(* CODESYS project EAS PLC.library
   Author: EAS
   Placeholder: EAS
   Title: EAS PLC
   Version: 1.0.0
   DefaultNamespace: EAS
   Company: ESCARRE AUTOMATIZACION Y SERVICIOS sl

Project tree, tasks and I/O mapping:
  libraries: Tc2_Standard, * (Beckhoff Automation GmbH); Tc2_System, * (Beckhoff Automation GmbH); Tc3_Module, * (Beckhoff Automation GmbH); Util, * (System)
  DUTs/
    data type TipusCurva
  GVLs/
    global variables GVL
  POUs/
    PLC/
      AddTanks/
        function block Circulation_TK [ST]
        function block Drain_TK [ST]
        function fCurvePerCen [ST]
        function block Introduction [ST]
        function block Introduction_M [ST]
      Elements/
        function block LiterCounter [ST]
        function block LitersPerLevel [ST]
        function block MeterCounter [ST]
        function block PulseTrain [ST]
        function block Washing_HT [ST]
      Fill/
        function block TemperatureFill [ST]
      Utils/
        AnalogConversions/
          function Canvi_Escala [ST]
          function Conv_Temp [ST]
        BitsConversions/
          function block Bits_to_Dword [ST]
          function block Bits_to_word [ST]
          function block Dword_to_bits [ST]
          function block Word_to_bits [ST]
        Counters/
          function block Calcul_Frequencia [ST]
          function block ContadorRapid [ST]
        FreqCycle/
          function block CalcFreq [ST]
          function block TCicle [ST]
        Timers/
          function block TMP [ST]
          function block TMPpausa [ST]
  VISUs/
*)

// DUTs/TipusCurva
TYPE TipusCurva :
STRUCT
	Table:ARRAY [0..10] OF point;
END_STRUCT
END_TYPE

// GVLs/GVL
VAR_GLOBAL RETAIN

(*=======================================	*)
(*		Curvas								*)
(*=======================================	*)

	CurvePerCent:ARRAY[0..19]OF TipusCurva;

END_VAR

// POUs/PLC/AddTanks/Circulation_TK
FUNCTION_BLOCK Circulation_TK
(*****************************************************************
Execute the recirculation of the add tank (Mac -> tank, tank -> mac) - 01/12/2021
v1.00
****************************************************************)
VAR_INPUT
	xActvRecirc:BOOL;				// Activate the function
	xPulsFinRecirc:BOOL;			// Finish the function
	xLowLevelRecirc:BOOL;			// Add tank Low level for the recirculation
	xHighLevelRecirc:BOOL;			// Add tank high level for the recirculation
	xMinimLevel:BOOL;				// Minimum tank level for the recirculation
	dwDrainTime:DWORD;				// Add tank drain time
END_VAR
VAR_OUTPUT
	xFiRecirc:BOOL;					// Recirculate finished
	xFill:BOOL;						// Add tank fill (runback)
	xIntro:BOOL;					// Add tank introduction (transfer)
END_VAR
VAR
	PararRecirculacio: BOOL;
	PararOmplerta: BOOL;
	OmplirEnRecirculacio: BOOL;
	PararIntroducio: BOOL;
	IntroduccioEnRecirculacio: BOOL;
	srPararRecirculacio : SR;
	TempoDescubrirNivBaix: TMP;
	Reircular: BOOL;
	FiBuidatCubeta: BOOL;
	BuidarCubeta: BOOL;
	TEmpoDrenatBuidat: TMP;
	srFiBuidatCubeta : SR;
END_VAR

// *********** Fin recircula por pulsador *****************
srPararRecirculacio(SET1:=xActvRecirc AND  xPulsFinRecirc, RESET:=NOT xActvRecirc , Q1=>PararRecirculacio );

Reircular := xActvRecirc AND NOT PararRecirculacio;

OmplirEnRecirculacio := Reircular AND NOT PararOmplerta;

IntroduccioEnRecirculacio := Reircular AND NOT PararIntroducio;
// ********* Pausa la introduccion si el nivel esta bajo *****************
TempoDescubrirNivBaix(xIN:=Reircular AND xLowLevelRecirc, dwSegons:=5 , xQ=> , dwTsegons=> );
PararIntroducio := NOT TempoDescubrirNivBaix.xQ; 

PararOmplerta := Reircular AND xHighLevelRecirc;

BuidarCubeta := xActvRecirc AND PararRecirculacio;

TEmpoDrenatBuidat(xIN:=BuidarCubeta AND NOT xMinimLevel, dwSegons:=dwDrainTime , xQ=> , dwTsegons=> );

srFiBuidatCubeta(SET1:=TEmpoDrenatBuidat.xQ , RESET:=NOT xActvRecirc , Q1=>FiBuidatCubeta );
// ************ Finaliza la recirculacion ********
xFiRecirc := FiBuidatCubeta;
// ************ Introduz a la maquina **********
xIntro := (BuidarCubeta AND NOT FiBuidatCubeta) OR IntroduccioEnRecirculacio;
// ************ Retorno de bano a la cubeta ********
xFill := OmplirEnRecirculacio;

END_FUNCTION_BLOCK

// POUs/PLC/AddTanks/Introduction
FUNCTION_BLOCK Introduction
(**********************************************************************
Control the transfering and dosing of the add tanks - 01/12/2021
v1.00
***********************************************************************)
VAR_INPUT
	xActvIntro:BOOL;			//Enable the function
	dwCurve:DWORD;				// Dosing curve
	dwTime:DWORD;				// Duration Time
	rLevel:REAL;				// Tank Level
	xLevelMin:BOOL;				// Tank Minimun Level
	xIniCond:BOOL;				// Initial condicions
	xPause:BOOL;				// Pause the function
END_VAR
VAR_OUTPUT
	xFiIntro:BOOL;				// End of the introduction
	rQTeoric:REAL;				// Teoric Quantity of the introduction (%)
	rQreal:REAL;				// Real Quantity of the introduction (%)
	xPrepareIntro:BOOL;			// Prepare an Introduction
	xDosIntro:BOOL;				// Introduct dosing (slow)
	xTransferIntro:BOOL;		// Introduct transfering (fast)
END_VAR
VAR
	IniciarIntro: BOOL;
	TEmpoInici: TMP;
	calculQt: CHARCURVE;
	rampatems: RAMP_REAL;
	tempsreal: REAL;
	Tempsensegons: REAL;
	IntroduccioDosificada: BOOL;
	IntroduccioDirecte: BOOL;
	TempsEnPercentatge: REAL;
	TaulaCurva:ARRAY [0..10]OF point;
	RampaTempsInt: INT;
	QteoricaINT: INT;
	ERROR: BYTE;
	entradaRampa: REAL;

	NivellInicial: REAL;
	TempsNivellinim: TMP;
	FiIntroDosificada: BOOL;
	TempsNivellinimDir: TMP;
	FiDirecte: BOOL;
	srFiIntro :SR;
END_VAR

// Inicia Intro
TEmpoInici(xIN:=xActvIntro AND xIniCond , dwSegons:=2 , xQ=>IniciarIntro , dwTsegons=> );

// Verifica si es introducion directa o dosificada
IF dwTime > 0
	THEN
		IntroduccioDosificada := TRUE;
		IntroduccioDirecte := FALSE;
	ELSE
		IntroduccioDosificada := FALSE;
		IntroduccioDirecte := TRUE;
END_IF

// Calculos del tiempo
Tempsensegons := DWORD_TO_REAL(dwTime*60);

IF IniciarIntro
	THEN
		EntradaRampa := Tempsensegons;
	ELSE
		EntradaRampa := 0;	
		NivellInicial := rLevel;
END_IF

// Si es introducin dosificada calcula la rampa
IF IntroduccioDosificada
	THEN
		rampatems(
			IN:= EntradaRampa, 
			ASCEND:= 1, 
			DESCEND:= Tempsensegons, 
			TIMEBASE:= T#1S, 
			RESET:= (IniciarIntro AND xPause) , 
			OUT=> tempsreal);

		TempsEnPercentatge := (tempsreal/Tempsensegons)*100;
END_IF

RampaTempsInt := REAL_TO_INT(TempsEnPercentatge*100);

TaulaCurva :=  fCurvePerCen(Curve:=DWORD_TO_INT (dwCurve));

calculQt(
	IN:= RampaTempsInt , 
	N:=11 , 
	P:=TaulaCurva , 
	OUT=>QteoricaINT , 
	ERR=>ERROR );

// Si se ha iniciado la introducion calcula el Qreal
IF IniciarIntro AND NivellInicial > 0
	THEN
		rQreal := (rLevel/NivellInicial)*100;
END_IF

rQTeoric := (INT_TO_REAL(QteoricaINT))/100;

xPrepareIntro := IniciarIntro AND NOT xFiIntro;

IF rQreal > rQTeoric AND IniciarIntro AND IntroduccioDosificada AND NOT xFiIntro
	THEN
		xDosIntro := TRUE;
	ELSE
		xDosIntro := FALSE;
END_IF

xTransferIntro := IntroduccioDosificada AND IniciarIntro AND NOT xFiIntro;

TempsNivellinim(xIN:=xLevelMin , dwSegons:=60 , xQ=> , dwTsegons=> );

IF rQTeoric <= 0 OR rQTeoric <= 0 OR TempsNivellinim.xQ OR IntroduccioDosificada OR IniciarIntro OR NOT xLevelMin
	THEN
		FiIntroDosificada := TRUE;
	ELSE
		FiIntroDosificada := FALSE;
END_IF

TempsNivellinimDir(xIN:= NOT xLevelMin , dwSegons:=3 , xQ=> , dwTsegons=> );

FiDirecte := NOT IntroduccioDosificada AND IniciarIntro AND TempsNivellinimDir.xQ;


srFiIntro(SET1:=(FiIntroDosificada OR FiDirecte) AND xActvIntro, RESET:= NOT xActvIntro , Q1=>xFiIntro);

END_FUNCTION_BLOCK

// POUs/PLC/AddTanks/fCurvePerCen
FUNCTION fCurvePerCen : ARRAY [0..10] OF POINT
(*******************************************************
Aquest Bloc Carrega per HardCode els valors de les les Corves percentuals.
Al demanar una corva retorna una taula de punts per a l'introduccio
=========================================
06/09/2006= Error corva7.
********************************************************)
VAR_INPUT
	Curve:INT;			// Curve (0 - 19)
END_VAR

VAR_OUTPUT

END_VAR	

VAR
END_VAR



(*Curve 0*)
GVL.CurvePerCent[0].Table[0].X:=0;
GVL.CurvePerCent[0].Table[0].Y:=10000;
GVL.CurvePerCent[0].Table[1].X:=1000;
GVL.CurvePerCent[0].Table[1].Y:=9000;
GVL.CurvePerCent[0].Table[2].X:=2000;
GVL.CurvePerCent[0].Table[2].Y:=8000;
GVL.CurvePerCent[0].Table[3].X:=3000;
GVL.CurvePerCent[0].Table[3].Y:=7000;
GVL.CurvePerCent[0].Table[4].X:=4000;
GVL.CurvePerCent[0].Table[4].Y:=6000;
GVL.CurvePerCent[0].Table[5].X:=5000;
GVL.CurvePerCent[0].Table[5].Y:=5000;
GVL.CurvePerCent[0].Table[6].X:=6000;
GVL.CurvePerCent[0].Table[6].Y:=4000;
GVL.CurvePerCent[0].Table[7].X:=7000;
GVL.CurvePerCent[0].Table[7].Y:=3000;
GVL.CurvePerCent[0].Table[8].X:=8000;
GVL.CurvePerCent[0].Table[8].Y:=2000;
GVL.CurvePerCent[0].Table[9].X:=9000;
GVL.CurvePerCent[0].Table[9].Y:=1000;
GVL.CurvePerCent[0].Table[10].X:=10000;
GVL.CurvePerCent[0].Table[10].Y:=0;

(*GVL.Curve 1*)
GVL.CurvePerCent[1].Table[0].X:=0;
GVL.CurvePerCent[1].Table[0].Y:=10000;
GVL.CurvePerCent[1].Table[1].X:=1000;
GVL.CurvePerCent[1].Table[1].Y:=9100;
GVL.CurvePerCent[1].Table[2].X:=2000;
GVL.CurvePerCent[1].Table[2].Y:=8200;
GVL.CurvePerCent[1].Table[3].X:=3000;
GVL.CurvePerCent[1].Table[3].Y:=7300;
GVL.CurvePerCent[1].Table[4].X:=4000;
GVL.CurvePerCent[1].Table[4].Y:=6400;
GVL.CurvePerCent[1].Table[5].X:=5000;
GVL.CurvePerCent[1].Table[5].Y:=5400;
GVL.CurvePerCent[1].Table[6].X:=6000;
GVL.CurvePerCent[1].Table[6].Y:=4500;
GVL.CurvePerCent[1].Table[7].X:=7000;
GVL.CurvePerCent[1].Table[7].Y:=3500;
GVL.CurvePerCent[1].Table[8].X:=8000;
GVL.CurvePerCent[1].Table[8].Y:=2400;
GVL.CurvePerCent[1].Table[9].X:=9000;
GVL.CurvePerCent[1].Table[9].Y:=1300;
GVL.CurvePerCent[1].Table[10].X:=10000;
GVL.CurvePerCent[1].Table[10].Y:=0;

(*GVL.Curve 2*)
GVL.CurvePerCent[2].Table[0].X:=0;
GVL.CurvePerCent[2].Table[0].Y:=10000;
GVL.CurvePerCent[2].Table[1].X:=1000;
GVL.CurvePerCent[2].Table[1].Y:=9200;
GVL.CurvePerCent[2].Table[2].X:=2000;
GVL.CurvePerCent[2].Table[2].Y:=8400;
GVL.CurvePerCent[2].Table[3].X:=3000;
GVL.CurvePerCent[2].Table[3].Y:=7600;
GVL.CurvePerCent[2].Table[4].X:=4000;
GVL.CurvePerCent[2].Table[4].Y:=6700;
GVL.CurvePerCent[2].Table[5].X:=5000;
GVL.CurvePerCent[2].Table[5].Y:=5800;
GVL.CurvePerCent[2].Table[6].X:=6000;
GVL.CurvePerCent[2].Table[6].Y:=4900;
GVL.CurvePerCent[2].Table[7].X:=7000;
GVL.CurvePerCent[2].Table[7].Y:=3900;
GVL.CurvePerCent[2].Table[8].X:=8000;
GVL.CurvePerCent[2].Table[8].Y:=2800;
GVL.CurvePerCent[2].Table[9].X:=9000;
GVL.CurvePerCent[2].Table[9].Y:=1500;
GVL.CurvePerCent[2].Table[10].X:=10000;
GVL.CurvePerCent[2].Table[10].Y:=0;

(*GVL.Curve 3*)
GVL.CurvePerCent[3].Table[0].X:=0;
GVL.CurvePerCent[3].Table[0].Y:=10000;
GVL.CurvePerCent[3].Table[1].X:=1000;
GVL.CurvePerCent[3].Table[1].Y:=9300;
GVL.CurvePerCent[3].Table[2].X:=2000;
GVL.CurvePerCent[3].Table[2].Y:=8500;
GVL.CurvePerCent[3].Table[3].X:=3000;
GVL.CurvePerCent[3].Table[3].Y:=7800;
GVL.CurvePerCent[3].Table[4].X:=4000;
GVL.CurvePerCent[3].Table[4].Y:=7000;
GVL.CurvePerCent[3].Table[5].X:=5000;
GVL.CurvePerCent[3].Table[5].Y:=6200;
GVL.CurvePerCent[3].Table[6].X:=6000;
GVL.CurvePerCent[3].Table[6].Y:=5300;
GVL.CurvePerCent[3].Table[7].X:=7000;
GVL.CurvePerCent[3].Table[7].Y:=4400;
GVL.CurvePerCent[3].Table[8].X:=8000;
GVL.CurvePerCent[3].Table[8].Y:=3200;
GVL.CurvePerCent[3].Table[9].X:=9000;
GVL.CurvePerCent[3].Table[9].Y:=1800;
GVL.CurvePerCent[3].Table[10].X:=10000;
GVL.CurvePerCent[3].Table[10].Y:=0;

(*GVL.Curve 4*)
GVL.CurvePerCent[4].Table[0].X:=0;
GVL.CurvePerCent[4].Table[0].Y:=10000;
GVL.CurvePerCent[4].Table[1].X:=1000;
GVL.CurvePerCent[4].Table[1].Y:=9400;
GVL.CurvePerCent[4].Table[2].X:=2000;
GVL.CurvePerCent[4].Table[2].Y:=8600;
GVL.CurvePerCent[4].Table[3].X:=3000;
GVL.CurvePerCent[4].Table[3].Y:=8100;
GVL.CurvePerCent[4].Table[4].X:=4000;
GVL.CurvePerCent[4].Table[4].Y:=7400;
GVL.CurvePerCent[4].Table[5].X:=5000;
GVL.CurvePerCent[4].Table[5].Y:=6600;
GVL.CurvePerCent[4].Table[6].X:=6000;
GVL.CurvePerCent[4].Table[6].Y:=5700;
GVL.CurvePerCent[4].Table[7].X:=7000;
GVL.CurvePerCent[4].Table[7].Y:=4900;
GVL.CurvePerCent[4].Table[8].X:=8000;
GVL.CurvePerCent[4].Table[8].Y:=3600;
GVL.CurvePerCent[4].Table[9].X:=9000;
GVL.CurvePerCent[4].Table[9].Y:=2100;
GVL.CurvePerCent[4].Table[10].X:=10000;
GVL.CurvePerCent[4].Table[10].Y:=0;

(*GVL.Curve 5*)
GVL.CurvePerCent[5].Table[0].X:=0;
GVL.CurvePerCent[5].Table[0].Y:=10000;
GVL.CurvePerCent[5].Table[1].X:=1000;
GVL.CurvePerCent[5].Table[1].Y:=9500;
GVL.CurvePerCent[5].Table[2].X:=2000;
GVL.CurvePerCent[5].Table[2].Y:=8800;
GVL.CurvePerCent[5].Table[3].X:=3000;
GVL.CurvePerCent[5].Table[3].Y:=8300;
GVL.CurvePerCent[5].Table[4].X:=4000;
GVL.CurvePerCent[5].Table[4].Y:=7600;
GVL.CurvePerCent[5].Table[5].X:=5000;
GVL.CurvePerCent[5].Table[5].Y:=7000;
GVL.CurvePerCent[5].Table[6].X:=6000;
GVL.CurvePerCent[5].Table[6].Y:=6200;
GVL.CurvePerCent[5].Table[7].X:=7000;
GVL.CurvePerCent[5].Table[7].Y:=5400;
GVL.CurvePerCent[5].Table[8].X:=8000;
GVL.CurvePerCent[5].Table[8].Y:=4000;
GVL.CurvePerCent[5].Table[9].X:=9000;
GVL.CurvePerCent[5].Table[9].Y:=2300;
GVL.CurvePerCent[5].Table[10].X:=10000;
GVL.CurvePerCent[5].Table[10].Y:=0;

(*GVL.Curve 6*)
GVL.CurvePerCent[6].Table[0].X:=0;
GVL.CurvePerCent[6].Table[0].Y:=10000;
GVL.CurvePerCent[6].Table[1].X:=1000;
GVL.CurvePerCent[6].Table[1].Y:=9500;
GVL.CurvePerCent[6].Table[2].X:=2000;
GVL.CurvePerCent[6].Table[2].Y:=9000;
GVL.CurvePerCent[6].Table[3].X:=3000;
GVL.CurvePerCent[6].Table[3].Y:=8500;
GVL.CurvePerCent[6].Table[4].X:=4000;
GVL.CurvePerCent[6].Table[4].Y:=8000;
GVL.CurvePerCent[6].Table[5].X:=5000;
GVL.CurvePerCent[6].Table[5].Y:=7400;
GVL.CurvePerCent[6].Table[6].X:=6000;
GVL.CurvePerCent[6].Table[6].Y:=6600;
GVL.CurvePerCent[6].Table[7].X:=7000;
GVL.CurvePerCent[6].Table[7].Y:=5800;
GVL.CurvePerCent[6].Table[8].X:=8000;
GVL.CurvePerCent[6].Table[8].Y:=4400;
GVL.CurvePerCent[6].Table[9].X:=9000;
GVL.CurvePerCent[6].Table[9].Y:=2600;
GVL.CurvePerCent[6].Table[10].X:=10000;
GVL.CurvePerCent[6].Table[10].Y:=0;

(*GVL.Curve 7*)
GVL.CurvePerCent[7].Table[0].X:=0;
GVL.CurvePerCent[7].Table[0].Y:=10000;
GVL.CurvePerCent[7].Table[1].X:=1000;
GVL.CurvePerCent[7].Table[1].Y:=9600;
GVL.CurvePerCent[7].Table[2].X:=2000;
GVL.CurvePerCent[7].Table[2].Y:=9200;
GVL.CurvePerCent[7].Table[3].X:=3000;
GVL.CurvePerCent[7].Table[3].Y:=8800;
GVL.CurvePerCent[7].Table[4].X:=4000;
GVL.CurvePerCent[7].Table[4].Y:=8300;
GVL.CurvePerCent[7].Table[5].X:=5000;
GVL.CurvePerCent[7].Table[5].Y:=7800;
GVL.CurvePerCent[7].Table[6].X:=6000;
GVL.CurvePerCent[7].Table[6].Y:=7100;
GVL.CurvePerCent[7].Table[7].X:=7000;
GVL.CurvePerCent[7].Table[7].Y:=6300;
GVL.CurvePerCent[7].Table[8].X:=8000;
GVL.CurvePerCent[7].Table[8].Y:=4800;
GVL.CurvePerCent[7].Table[9].X:=9000;
GVL.CurvePerCent[7].Table[9].Y:=2800;
GVL.CurvePerCent[7].Table[10].X:=10000;
GVL.CurvePerCent[7].Table[10].Y:=0;

(*GVL.Curve 8*)
GVL.CurvePerCent[8].Table[0].X:=0;
GVL.CurvePerCent[8].Table[0].Y:=10000;
GVL.CurvePerCent[8].Table[1].X:=1000;
GVL.CurvePerCent[8].Table[1].Y:=9700;
GVL.CurvePerCent[8].Table[2].X:=2000;
GVL.CurvePerCent[8].Table[2].Y:=9400;
GVL.CurvePerCent[8].Table[3].X:=3000;
GVL.CurvePerCent[8].Table[3].Y:=9100;
GVL.CurvePerCent[8].Table[4].X:=4000;
GVL.CurvePerCent[8].Table[4].Y:=8600;
GVL.CurvePerCent[8].Table[5].X:=5000;
GVL.CurvePerCent[8].Table[5].Y:=8200;
GVL.CurvePerCent[8].Table[6].X:=6000;
GVL.CurvePerCent[8].Table[6].Y:=7500;
GVL.CurvePerCent[8].Table[7].X:=7000;
GVL.CurvePerCent[8].Table[7].Y:=6700;
GVL.CurvePerCent[8].Table[8].X:=8000;
GVL.CurvePerCent[8].Table[8].Y:=5200;
GVL.CurvePerCent[8].Table[9].X:=9000;
GVL.CurvePerCent[8].Table[9].Y:=3100;
GVL.CurvePerCent[8].Table[10].X:=10000;
GVL.CurvePerCent[8].Table[10].Y:=0;

(*GVL.Curve 9*)
GVL.CurvePerCent[9].Table[0].X:=0;
GVL.CurvePerCent[9].Table[0].Y:=10000;
GVL.CurvePerCent[9].Table[1].X:=1000;
GVL.CurvePerCent[9].Table[1].Y:=9800;
GVL.CurvePerCent[9].Table[2].X:=2000;
GVL.CurvePerCent[9].Table[2].Y:=9600;
GVL.CurvePerCent[9].Table[3].X:=3000;
GVL.CurvePerCent[9].Table[3].Y:=9300;
GVL.CurvePerCent[9].Table[4].X:=4000;
GVL.CurvePerCent[9].Table[4].Y:=9000;
GVL.CurvePerCent[9].Table[5].X:=5000;
GVL.CurvePerCent[9].Table[5].Y:=8600;
GVL.CurvePerCent[9].Table[6].X:=6000;
GVL.CurvePerCent[9].Table[6].Y:=7900;
GVL.CurvePerCent[9].Table[7].X:=7000;
GVL.CurvePerCent[9].Table[7].Y:=7100;
GVL.CurvePerCent[9].Table[8].X:=8000;
GVL.CurvePerCent[9].Table[8].Y:=5600;
GVL.CurvePerCent[9].Table[9].X:=9000;
GVL.CurvePerCent[9].Table[9].Y:=3400;
GVL.CurvePerCent[9].Table[10].X:=10000;
GVL.CurvePerCent[9].Table[10].Y:=0;

(*GVL.Curve 10*)
GVL.CurvePerCent[10].Table[0].X:=0;
GVL.CurvePerCent[10].Table[0].Y:=10000;
GVL.CurvePerCent[10].Table[1].X:=1000;
GVL.CurvePerCent[10].Table[1].Y:=9000;
GVL.CurvePerCent[10].Table[2].X:=2000;
GVL.CurvePerCent[10].Table[2].Y:=8000;
GVL.CurvePerCent[10].Table[3].X:=3000;
GVL.CurvePerCent[10].Table[3].Y:=7000;
GVL.CurvePerCent[10].Table[4].X:=4000;
GVL.CurvePerCent[10].Table[4].Y:=6000;
GVL.CurvePerCent[10].Table[5].X:=5000;
GVL.CurvePerCent[10].Table[5].Y:=5000;
GVL.CurvePerCent[10].Table[6].X:=6000;
GVL.CurvePerCent[10].Table[6].Y:=4000;
GVL.CurvePerCent[10].Table[7].X:=7000;
GVL.CurvePerCent[10].Table[7].Y:=3000;
GVL.CurvePerCent[10].Table[8].X:=8000;
GVL.CurvePerCent[10].Table[8].Y:=2000;
GVL.CurvePerCent[10].Table[9].X:=9000;
GVL.CurvePerCent[10].Table[9].Y:=1000;
GVL.CurvePerCent[10].Table[10].X:=10000;
GVL.CurvePerCent[10].Table[10].Y:=0;

(*GVL.Curve 11*)
GVL.CurvePerCent[11].Table[0].X:=0;
GVL.CurvePerCent[11].Table[0].Y:=10000;
GVL.CurvePerCent[11].Table[1].X:=1000;
GVL.CurvePerCent[11].Table[1].Y:=8700;
GVL.CurvePerCent[11].Table[2].X:=2000;
GVL.CurvePerCent[11].Table[2].Y:=7600;
GVL.CurvePerCent[11].Table[3].X:=3000;
GVL.CurvePerCent[11].Table[3].Y:=6500;
GVL.CurvePerCent[11].Table[4].X:=4000;
GVL.CurvePerCent[11].Table[4].Y:=5500;
GVL.CurvePerCent[11].Table[5].X:=5000;
GVL.CurvePerCent[11].Table[5].Y:=4600;
GVL.CurvePerCent[11].Table[6].X:=6000;
GVL.CurvePerCent[11].Table[6].Y:=3600;
GVL.CurvePerCent[11].Table[7].X:=7000;
GVL.CurvePerCent[11].Table[7].Y:=2700;
GVL.CurvePerCent[11].Table[8].X:=8000;
GVL.CurvePerCent[11].Table[8].Y:=1800;
GVL.CurvePerCent[11].Table[9].X:=9000;
GVL.CurvePerCent[11].Table[9].Y:=900;
GVL.CurvePerCent[11].Table[10].X:=10000;
GVL.CurvePerCent[11].Table[10].Y:=0;

(*GVL.Curve 12*)
GVL.CurvePerCent[12].Table[0].X:=0;
GVL.CurvePerCent[12].Table[0].Y:=10000;
GVL.CurvePerCent[12].Table[1].X:=1000;
GVL.CurvePerCent[12].Table[1].Y:=8500;
GVL.CurvePerCent[12].Table[2].X:=2000;
GVL.CurvePerCent[12].Table[2].Y:=7200;
GVL.CurvePerCent[12].Table[3].X:=3000;
GVL.CurvePerCent[12].Table[3].Y:=6100;
GVL.CurvePerCent[12].Table[4].X:=4000;
GVL.CurvePerCent[12].Table[4].Y:=5100;
GVL.CurvePerCent[12].Table[5].X:=5000;
GVL.CurvePerCent[12].Table[5].Y:=4200;
GVL.CurvePerCent[12].Table[6].X:=6000;
GVL.CurvePerCent[12].Table[6].Y:=3300;
GVL.CurvePerCent[12].Table[7].X:=7000;
GVL.CurvePerCent[12].Table[7].Y:=2400;
GVL.CurvePerCent[12].Table[8].X:=8000;
GVL.CurvePerCent[12].Table[8].Y:=1600;
GVL.CurvePerCent[12].Table[9].X:=9000;
GVL.CurvePerCent[12].Table[9].Y:=800;
GVL.CurvePerCent[12].Table[10].X:=10000;
GVL.CurvePerCent[12].Table[10].Y:=0;

(*GVL.Curve 13*)
GVL.CurvePerCent[13].Table[0].X:=0;
GVL.CurvePerCent[13].Table[0].Y:=10000;
GVL.CurvePerCent[13].Table[1].X:=1000;
GVL.CurvePerCent[13].Table[1].Y:=8200;
GVL.CurvePerCent[13].Table[2].X:=2000;
GVL.CurvePerCent[13].Table[2].Y:=6800;
GVL.CurvePerCent[13].Table[3].X:=3000;
GVL.CurvePerCent[13].Table[3].Y:=5600;
GVL.CurvePerCent[13].Table[4].X:=4000;
GVL.CurvePerCent[13].Table[4].Y:=4700;
GVL.CurvePerCent[13].Table[5].X:=5000;
GVL.CurvePerCent[13].Table[5].Y:=3800;
GVL.CurvePerCent[13].Table[6].X:=6000;
GVL.CurvePerCent[13].Table[6].Y:=3000;
GVL.CurvePerCent[13].Table[7].X:=7000;
GVL.CurvePerCent[13].Table[7].Y:=2200;
GVL.CurvePerCent[13].Table[8].X:=8000;
GVL.CurvePerCent[13].Table[8].Y:=1500;
GVL.CurvePerCent[13].Table[9].X:=9000;
GVL.CurvePerCent[13].Table[9].Y:=700;
GVL.CurvePerCent[13].Table[10].X:=10000;
GVL.CurvePerCent[13].Table[10].Y:=0;

(*GVL.Curve 14*)
GVL.CurvePerCent[14].Table[0].X:=0;
GVL.CurvePerCent[14].Table[0].Y:=10000;
GVL.CurvePerCent[14].Table[1].X:=1000;
GVL.CurvePerCent[14].Table[1].Y:=7900;
GVL.CurvePerCent[14].Table[2].X:=2000;
GVL.CurvePerCent[14].Table[2].Y:=6400;
GVL.CurvePerCent[14].Table[3].X:=3000;
GVL.CurvePerCent[14].Table[3].Y:=5100;
GVL.CurvePerCent[14].Table[4].X:=4000;
GVL.CurvePerCent[14].Table[4].Y:=4300;
GVL.CurvePerCent[14].Table[5].X:=5000;
GVL.CurvePerCent[14].Table[5].Y:=3400;
GVL.CurvePerCent[14].Table[6].X:=6000;
GVL.CurvePerCent[14].Table[6].Y:=2600;
GVL.CurvePerCent[14].Table[7].X:=5000;
GVL.CurvePerCent[14].Table[7].Y:=1900;
GVL.CurvePerCent[14].Table[8].X:=8000;
GVL.CurvePerCent[14].Table[8].Y:=1400;
GVL.CurvePerCent[14].Table[9].X:=9000;
GVL.CurvePerCent[14].Table[9].Y:=600;
GVL.CurvePerCent[14].Table[10].X:=10000;
GVL.CurvePerCent[14].Table[10].Y:=0;

(*GVL.Curve 15*)
GVL.CurvePerCent[15].Table[0].X:=0;
GVL.CurvePerCent[15].Table[0].Y:=10000;
GVL.CurvePerCent[15].Table[1].X:=1000;
GVL.CurvePerCent[15].Table[1].Y:=7700;
GVL.CurvePerCent[15].Table[2].X:=2000;
GVL.CurvePerCent[15].Table[2].Y:=6000;
GVL.CurvePerCent[15].Table[3].X:=3000;
GVL.CurvePerCent[15].Table[3].Y:=4600;
GVL.CurvePerCent[15].Table[4].X:=4000;
GVL.CurvePerCent[15].Table[4].Y:=3800;
GVL.CurvePerCent[15].Table[5].X:=5000;
GVL.CurvePerCent[15].Table[5].Y:=3000;
GVL.CurvePerCent[15].Table[6].X:=6000;
GVL.CurvePerCent[15].Table[6].Y:=2400;
GVL.CurvePerCent[15].Table[7].X:=7000;
GVL.CurvePerCent[15].Table[7].Y:=1700;
GVL.CurvePerCent[15].Table[8].X:=8000;
GVL.CurvePerCent[15].Table[8].Y:=1200;
GVL.CurvePerCent[15].Table[9].X:=9000;
GVL.CurvePerCent[15].Table[9].Y:=500;
GVL.CurvePerCent[15].Table[10].X:=10000;
GVL.CurvePerCent[15].Table[10].Y:=0;

(*GVL.Curve 16*)
GVL.CurvePerCent[16].Table[0].X:=0;
GVL.CurvePerCent[16].Table[0].Y:=10000;
GVL.CurvePerCent[16].Table[1].X:=1000;
GVL.CurvePerCent[16].Table[1].Y:=7400;
GVL.CurvePerCent[16].Table[2].X:=2000;
GVL.CurvePerCent[16].Table[2].Y:=5600;
GVL.CurvePerCent[16].Table[3].X:=3000;
GVL.CurvePerCent[16].Table[3].Y:=4200;
GVL.CurvePerCent[16].Table[4].X:=4000;
GVL.CurvePerCent[16].Table[4].Y:=3400;
GVL.CurvePerCent[16].Table[5].X:=5000;
GVL.CurvePerCent[16].Table[5].Y:=2600;
GVL.CurvePerCent[16].Table[6].X:=6000;
GVL.CurvePerCent[16].Table[6].Y:=2000;
GVL.CurvePerCent[16].Table[7].X:=7000;
GVL.CurvePerCent[16].Table[7].Y:=1500;
GVL.CurvePerCent[16].Table[8].X:=8000;
GVL.CurvePerCent[16].Table[8].Y:=1000;
GVL.CurvePerCent[16].Table[9].X:=9000;
GVL.CurvePerCent[16].Table[9].Y:=500;
GVL.CurvePerCent[16].Table[10].X:=10000;
GVL.CurvePerCent[16].Table[10].Y:=0;

(*GVL.Curve 17*)
GVL.CurvePerCent[17].Table[0].X:=0;
GVL.CurvePerCent[17].Table[0].Y:=10000;
GVL.CurvePerCent[17].Table[1].X:=1000;
GVL.CurvePerCent[17].Table[1].Y:=7200;
GVL.CurvePerCent[17].Table[2].X:=2000;
GVL.CurvePerCent[17].Table[2].Y:=5200;
GVL.CurvePerCent[17].Table[3].X:=3000;
GVL.CurvePerCent[17].Table[3].Y:=3700;
GVL.CurvePerCent[17].Table[4].X:=4000;
GVL.CurvePerCent[17].Table[4].Y:=2900;
GVL.CurvePerCent[17].Table[5].X:=5000;
GVL.CurvePerCent[17].Table[5].Y:=2200;
GVL.CurvePerCent[17].Table[6].X:=6000;
GVL.CurvePerCent[17].Table[6].Y:=1700;
GVL.CurvePerCent[17].Table[7].X:=7000;
GVL.CurvePerCent[17].Table[7].Y:=1200;
GVL.CurvePerCent[17].Table[8].X:=8000;
GVL.CurvePerCent[17].Table[8].Y:=800;
GVL.CurvePerCent[17].Table[9].X:=9000;
GVL.CurvePerCent[17].Table[9].Y:=400;
GVL.CurvePerCent[17].Table[10].X:=10000;
GVL.CurvePerCent[17].Table[10].Y:=0;

(*GVL.Curve 18*)
GVL.CurvePerCent[18].Table[0].X:=0;
GVL.CurvePerCent[18].Table[0].Y:=10000;
GVL.CurvePerCent[18].Table[1].X:=1000;
GVL.CurvePerCent[18].Table[1].Y:=6900;
GVL.CurvePerCent[18].Table[2].X:=2000;
GVL.CurvePerCent[18].Table[2].Y:=4800;
GVL.CurvePerCent[18].Table[3].X:=3000;
GVL.CurvePerCent[18].Table[3].Y:=3300;
GVL.CurvePerCent[18].Table[4].X:=4000;
GVL.CurvePerCent[18].Table[4].Y:=2500;
GVL.CurvePerCent[18].Table[5].X:=5000;
GVL.CurvePerCent[18].Table[5].Y:=1800;
GVL.CurvePerCent[18].Table[6].X:=6000;
GVL.CurvePerCent[18].Table[6].Y:=1400;
GVL.CurvePerCent[18].Table[7].X:=7000;
GVL.CurvePerCent[18].Table[7].Y:=900;
GVL.CurvePerCent[18].Table[8].X:=8000;
GVL.CurvePerCent[18].Table[8].Y:=600;
GVL.CurvePerCent[18].Table[9].X:=9000;
GVL.CurvePerCent[18].Table[9].Y:=300;
GVL.CurvePerCent[18].Table[10].X:=10000;
GVL.CurvePerCent[18].Table[10].Y:=0;

(*GVL.Curve 19*)
GVL.CurvePerCent[19].Table[0].X:=0;
GVL.CurvePerCent[19].Table[0].Y:=10000;
GVL.CurvePerCent[19].Table[1].X:=1000;
GVL.CurvePerCent[19].Table[1].Y:=6600;
GVL.CurvePerCent[19].Table[2].X:=2000;
GVL.CurvePerCent[19].Table[2].Y:=4400;
GVL.CurvePerCent[19].Table[3].X:=3000;
GVL.CurvePerCent[19].Table[3].Y:=2900;
GVL.CurvePerCent[19].Table[4].X:=4000;
GVL.CurvePerCent[19].Table[4].Y:=1900;
GVL.CurvePerCent[19].Table[5].X:=5000;
GVL.CurvePerCent[19].Table[5].Y:=1400;
GVL.CurvePerCent[19].Table[6].X:=6000;
GVL.CurvePerCent[19].Table[6].Y:=1000;
GVL.CurvePerCent[19].Table[7].X:=7000;
GVL.CurvePerCent[19].Table[7].Y:=700;
GVL.CurvePerCent[19].Table[8].X:=8000;
GVL.CurvePerCent[19].Table[8].Y:=400;
GVL.CurvePerCent[19].Table[9].X:=9000;
GVL.CurvePerCent[19].Table[9].Y:=200;
GVL.CurvePerCent[19].Table[10].X:=10000;
GVL.CurvePerCent[19].Table[10].Y:=0;


(*************************************************************************************************)
(*	Cargar Curve	*)

fCurvePerCen:=CurvePerCent[Curve].Table;

END_FUNCTION

// POUs/PLC/Utils/Timers/TMP
FUNCTION_BLOCK TMP
(**********************************************************
Timer in seconds with a DWORD input - 29/11/2021
V1.0
*********************************************************)
VAR_INPUT
	xIN:BOOL;			// Enable Input
	dwSegons:DWORD;		// Setpoint Time (seconds) Input
END_VAR
VAR_OUTPUT
	xQ:BOOL;					// Boolean Output
	dwTsegons:DWORD;			// Currently Time (seconds) Output
END_VAR

VAR
	TEmporitz: TON;
	Temps: TIME;
	TempsTrans: TIME;
END_VAR

Temps := REAL_TO_TIME (DWORD_TO_REAL (dwSegons)*1000);

TEmporitz(IN:=xIN , PT:=Temps , Q=>xQ , ET=>TempsTrans );

dwTsegons := REAL_TO_DWORD(TIME_TO_REAL (TempsTrans)/1000);

END_FUNCTION_BLOCK

// POUs/PLC/AddTanks/Drain_TK
FUNCTION_BLOCK Drain_TK 
(*************************************************************++
Execute the washing and drain of an add tank.
Available drain options:
type=0 => all the washings (2 to machine + 1 to the drain), 
type=1 => 1 to the machine,
type=2 => 2 to the machine,
type=3 => (2 to machine + 1 to the drain), 
01/12/2021
V1.00
*******************************************************************)
VAR_INPUT
	xStartWash:BOOL;			// Enable function input
	xMinimLevel:BOOL;			// Minimum Level Input
	dwDetectLowLevelTime:DWORD;	// Delay to detect the low level
	dwDrainTime:DWORD;			// Drain Time
	dw1stWashTime:DWORD;		// 1st Wash Time
	dw2ndWashTime:DWORD;		// 2nd Wash Time
	dw3rdWashTime:DWORD;		// 3rd Wash Time
	DrainType:DWORD;			// Drain Option (0 - 3)
END_VAR

VAR_OUTPUT
	xFinWash:BOOL;				// Function finished			
	xWash:BOOL;					// Fill the add tank output
	xToMachine:BOOL;			// Transfer add tank to machine
	xToDrain:BOOL;				// Drain add tank
END_VAR

VAR
	FerTotsElsRentats: BOOL;
	NomesRentatsAMaquina: BOOL;
	NoFerRentats: BOOL;
	FiPrimerRentat: BOOL;
	PrimerRentat: BOOL;
	TempoPrimerRentat: TMP;
	FiPrimerBuidat: BOOL;
	PrimerBuidat: BOOL;
	FiSegonRentat: BOOL;
	SegonRentat: BOOL;
	FiSegonBuidat: BOOL;
	SegonBuidat: BOOL;
	TempoPrimerBuidat: TMP;
	TempoSegonRentat: TMP;
	TempoSegonBuidat: TMP;
	TempoTercerRentat: TMP;
	TempoTercerBuidat: TMP;
	FiTercerRentat: BOOL;
	TercerRentat: BOOL;
	FiTercerBuidat: BOOL;
	TercerBuidat: BOOL;
	TempoBuit: TMP;
	ComencaArentar: BOOL;
	BuidaDelTot: BOOL;
	srComencaArentar : SR;
	srFiPrimerRentat : SR;
	srFiPrimerBuidat : SR;
	srFiSegonRentat  : SR;
	srFiSegonBuidat  : SR;
	srFiTercerRentat : SR;
	srFiTercerBuidat : SR;
END_VAR

// ********** Define el tipo de lavado ***********
CASE DrainType OF
	0 : FerTotsElsRentats := TRUE;
		NoFerRentats := FALSE;
		NomesRentatsAMaquina := FALSE;
	1 : FerTotsElsRentats := FALSE;
		NoFerRentats := TRUE;
		NomesRentatsAMaquina := FALSE;
	2 : FerTotsElsRentats := FALSE;
		NoFerRentats := FALSE;
		NomesRentatsAMaquina := TRUE;
	3 : FerTotsElsRentats := TRUE;
		NoFerRentats := FALSE;
		NomesRentatsAMaquina := FALSE;
END_CASE

// ************** Empeza el lavado **************
TempoBuit(xIN:=xStartWash AND NOT  xMinimLevel, dwSegons:=2 , xQ=> , dwTsegons=> );
srComencaArentar(SET1:=TempoBuit.xQ , RESET:= NOT xStartWash , Q1=>ComencaArentar );

BuidaDelTot := xStartWash AND NOT ComencaArentar;

// ********** Control Primer Lavado ******************
PrimerRentat := ComencaArentar AND NOT FiPrimerRentat;

TempoPrimerRentat(xIN:=ComencaArentar , dwSegons:=dw1stWashTime , xQ=> , dwTsegons=> );
srFiPrimerRentat(SET1:=TempoPrimerRentat.xQ , RESET:= NOT xStartWash , Q1=>FiPrimerRentat );

PrimerBuidat := FiPrimerRentat AND NOT FiPrimerBuidat;

TempoPrimerBuidat(xIN:=PrimerBuidat AND NOT  xMinimLevel, dwSegons:=dwDetectLowLevelTime , xQ=> , dwTsegons=> );
srFiPrimerBuidat(SET1:=TempoPrimerBuidat.xQ , RESET:=NOT xStartWash  , Q1=>FiPrimerBuidat );

// ********** Control Segun Lavado ***************** 
SegonRentat := FiPrimerBuidat AND NOT FiSegonRentat;

TempoSegonRentat(xIN:=SegonRentat , dwSegons:=dw2ndWashTime , xQ=> , dwTsegons=> );
srFiSegonRentat(SET1:=TempoSegonRentat.xQ , RESET:=NOT xStartWash  , Q1=>FiSegonRentat );

SegonBuidat := FiSegonRentat AND NOT FiSegonBuidat;

TempoSegonBuidat(xIN:=SegonBuidat AND NOT xMinimLevel, dwSegons:=dwDetectLowLevelTime , xQ=> , dwTsegons=> );
srFiSegonBuidat(SET1:=TempoSegonBuidat.xQ , RESET:=NOT xStartWash  , Q1=>FiSegonBuidat );

// ********** Control Tercer Lavado ***************** 
TercerRentat := FiSegonBuidat AND NOT FiTercerRentat;

TempoTercerRentat(xIN:=TercerRentat , dwSegons:=dw3rdWashTime , xQ=> , dwTsegons=> );
srFiTercerRentat(SET1:=TempoTercerRentat.xQ , RESET:=NOT xStartWash  , Q1=>FiTercerRentat );

TercerBuidat := FiTercerRentat AND NOT FiTercerBuidat;

TempoTercerBuidat(xIN:=TercerBuidat AND NOT xMinimLevel, dwSegons:=dwDrainTime , xQ=> , dwTsegons=> );
srFiTercerBuidat(SET1:=TempoTercerBuidat.xQ , RESET:=NOT xStartWash  , Q1=>FiTercerBuidat);

// ************* Finaliza los lavados ****************
xFinWash := xStartWash AND ((FerTotsElsRentats AND FiTercerBuidat) OR (NomesRentatsAMaquina AND FiSegonBuidat) OR (NoFerRentats AND FiPrimerBuidat));

// ************** Activa salidas *************
xWash	:= xStartWash AND (PrimerRentat OR SegonRentat OR TercerRentat);

xToMachine := NOT xFinWash AND (PrimerBuidat OR SegonBuidat OR BuidaDelTot);

xToDrain := NOT xFinWash AND TercerBuidat;

END_FUNCTION_BLOCK

// POUs/PLC/AddTanks/Introduction_M
FUNCTION_BLOCK Introduction_M
(**********************************************************************
Control the transfering and dosing of the add tanks with proportional valve
- 01/12/2021
v1.00
***********************************************************************)
VAR_INPUT
	xActvIntro:BOOL;			//Enable the function
	dwCurve:DWORD;				// Dosing curve
	dwTime:DWORD;				// Duration Time
	rLevel:REAL;				// Tank Level
	xLevelMin:BOOL;				// Tank Minimun Level
	xIniCond:BOOL;				// Initial condicions
	xPause:BOOL;				// Pause the function
	rPro: REAL;					// PID - P
	rInt: REAL;					// PID - I
	rDer: REAL;					// PID - D
END_VAR
VAR_OUTPUT
	xFiIntro:BOOL;				// End of the introduction
	rQTeoric:REAL;				// Teoric Quantity of the introduction (%)
	rQreal:REAL;				// Real Quantity of the introduction (%)
	xPrepareIntro:BOOL;			// Prepare an Introduction
	xDosIntro:BOOL;				// Introduct dosing (slow)
	xTransferIntro:BOOL;		// Introduct transfering (fast)
	rProportionalValve:REAL;	// % open proportiuonal valve
END_VAR
VAR
	IniciarIntro: BOOL;
	TEmpoInici: TMP;

	calculQt: CHARCURVE;
	rampatems: RAMP_REAL;
	tempsreal: REAL;
	Tempsensegons: REAL;

	IntroduccioDosificada: BOOL;
	IntroduccioDirecte: BOOL;
	TempsEnPercentatge: REAL;
	TaulaCurva:ARRAY [0..10]OF point;
	RampaTempsInt: INT;
	QteoricaINT: INT;
	ERROR: BYTE;
	entradaRampa: REAL;
	NivellInicial: REAL;
	TempsNivellinim: TMP;
	FiIntroDosificada: BOOL;
	TempsNivellinimDir: TMP;
	FiDirecte: BOOL;
	AperturaValvRegulant: PID;
	srFiIntro :SR;
	APERTURApid: REAL;
END_VAR

// *********** Inicia Intro ********************
TEmpoInici(xIN:=xActvIntro AND xIniCond , dwSegons:=2 , xQ=>IniciarIntro , dwTsegons=> );

// ************ Verifica si es introducion directa o dosificada *****************
IF dwTime > 0
	THEN
		IntroduccioDosificada := TRUE;
		IntroduccioDirecte := FALSE;
	ELSE
		IntroduccioDosificada := FALSE;
		IntroduccioDirecte := TRUE;
END_IF

// *************** Calculos del tiempo **********************
Tempsensegons := DWORD_TO_REAL(dwTime*60);

IF IniciarIntro
	THEN
		EntradaRampa := Tempsensegons;
	ELSE
		EntradaRampa := 0;	
		NivellInicial := rLevel;
END_IF

// ************* Si es introducin dosificada calcula la rampa *************
IF IntroduccioDosificada
	THEN
		rampatems(
			IN:= EntradaRampa, 
			ASCEND:= 1, 
			DESCEND:= Tempsensegons, 
			TIMEBASE:= T#1S, 
			RESET:= (IniciarIntro AND xPause) , 
			OUT=> tempsreal);

		TempsEnPercentatge := (tempsreal/Tempsensegons)*100;
END_IF

RampaTempsInt := REAL_TO_INT(TempsEnPercentatge*100);

TaulaCurva :=  fCurvePerCen(Curve:=DWORD_TO_INT (dwCurve));

calculQt(
	IN:= RampaTempsInt , 
	N:=11 , 
	P:=TaulaCurva , 
	OUT=>QteoricaINT , 
	ERR=>ERROR );

// **************** Si se ha iniciado la introducion calcula el Qreal *************
IF IniciarIntro AND NivellInicial > 0
	THEN
		rQreal := (rLevel/NivellInicial)*100;
END_IF

rQTeoric := (INT_TO_REAL(QteoricaINT))/100;

xPrepareIntro := IniciarIntro AND NOT xFiIntro;

xDosIntro := IntroduccioDosificada AND IniciarIntro AND NOT xFiIntro;

xTransferIntro := IntroduccioDirecte AND IniciarIntro AND NOT xFiIntro;

TempsNivellinim(xIN:=xLevelMin , dwSegons:=60 , xQ=> , dwTsegons=> );

IF (rQTeoric <= 0 OR rQTeoric <= 0 OR TempsNivellinim.xQ) AND IntroduccioDosificada AND IniciarIntro
	THEN
		FiIntroDosificada := TRUE;
	ELSE
		FiIntroDosificada := FALSE;
END_IF

TempsNivellinimDir(xIN:= NOT xLevelMin , dwSegons:=3 , xQ=> , dwTsegons=> );

FiDirecte := NOT IntroduccioDosificada AND IniciarIntro AND TempsNivellinimDir.xQ;

srFiIntro(SET1:=(FiIntroDosificada OR FiDirecte) AND xActvIntro, RESET:= NOT xActvIntro , Q1=>xFiIntro);

// ************** Regula la apertura de la valvula modulante ****************
AperturaValvRegulant(
	ACTUAL:= 100-rQreal, 
	SET_POINT:= 100-rQTeoric, 
	KP:= rPro, 
	TN:= rInt, 
	TV:= rDer, 
	Y_MANUAL:= , 
	Y_OFFSET:= , 
	Y_MIN:= 0, 
	Y_MAX:= 100, 
	MANUAL:= , 
	RESET:= NOT xDosIntro OR AperturaValvRegulant.OVERFLOW , 
	Y=> rProportionalValve, 
	LIMITS_ACTIVE=> , 
	OVERFLOW=> );

END_FUNCTION_BLOCK

// POUs/PLC/Elements/LiterCounter
FUNCTION_BLOCK LiterCounter
(*************************************************************
Convert a flow input into liters - 01/12/2021
V1.00
*************************************************************)
VAR_INPUT
	xActive : BOOL;			// Active the function
	rFlow :   REAL;			// Flow Input (l/min)
END_VAR
VAR_OUTPUT
	rLiters :   REAL;		// Liter output (REAL)
	dwLiters : 	DWORD;		//	Liter output (DDWORD)
END_VAR
VAR
	LitersSum : REAL;
	Periodecicle:Tcicle;
	ov: BOOL;
	INTEG: INTEGRAL;	
END_VAR


INTEG(
	IN:=rFlow , 
	TM:=10 , 
	RESET:=ov OR NOT xActive , 
	OUT=> LitersSum, 
	OVERFLOW=>ov );
	
rLiters := LitersSum/60;
dwLiters := REAL_TO_DWORD(LitersSum/60);

END_FUNCTION_BLOCK

// POUs/PLC/Utils/FreqCycle/TCicle
FUNCTION_BLOCK Tcicle
(**********************************************************
 - 29/11/2021
V1.00
*********************************************************)
VAR_INPUT

END_VAR
VAR_OUTPUT
	dwPeriode_Cicle:DWORD;		// Cycle Peryod
END_VAR

VAR_IN_OUT

END_VAR

VAR
	tempo: TON;
	reset: BOOL;
	t_actual: TIME;
	t_anterior: TIME;
	Periode: TIME;
END_VAR

tempo(IN:=NOT reset , PT:=T#7D , Q=>reset , ET=>t_actual );

Periode:= T_actual-T_anterior;

IF	NOT reset
	THEN
		T_anterior := T_actual;
END_IF

dwPeriode_cicle := TIME_TO_DWORD(Periode);

END_FUNCTION_BLOCK

// POUs/PLC/Elements/LitersPerLevel
FUNCTION_BLOCK LitersPerLevel
(**********************************************
Convert an Level input into Liters - 01/12/2021
V1.00
***********************************************)
VAR_INPUT
	rLevel:REAL;
	dwN0:DWORD;
	dwN10:DWORD;
	dwN20:DWORD;
	dwN30:DWORD;
	dwN40:DWORD;
	dwN50:DWORD;
	dwN60:DWORD;
	dwN70:DWORD;
	dwN80:DWORD;
	dwN90:DWORD;
	dwN100:DWORD;
END_VAR
VAR_OUTPUT
	rLiters:REAL;
END_VAR
VAR
	iLiters:INT;
	LitrosMaq: CHARCURVE;
	litrosNivell:ARRAY[0..10]OF point;
END_VAR


litrosNivell[0].X := 0;
litrosNivell[0].Y := dwN0;
litrosNivell[1].X := 100;
litrosNivell[1].Y := dwN10;
litrosNivell[2].X := 200;
litrosNivell[2].Y := dwN20;
litrosNivell[3].X := 300; 
litrosNivell[3].Y := dwN30;
litrosNivell[4].X := 400;
litrosNivell[4].Y := dwN40;
litrosNivell[5].X := 500;
litrosNivell[5].Y := dwN50;
litrosNivell[6].X := 600;
litrosNivell[6].Y := dwN60;
litrosNivell[7].X := 700;
litrosNivell[7].Y := dwN70;
litrosNivell[8].X := 800;
litrosNivell[8].Y := dwN80;
litrosNivell[9].X := 900;
litrosNivell[9].Y := dwN90;
litrosNivell[10].X := 1000;
litrosNivell[10].Y := dwN100;

LitrosMaq(
	IN:= REAL_TO_INT(rLevel*10) , 
	N:= 11, 
	P:= litrosNivell, 
	OUT=> iLiters, 
	ERR=> );

rLiters := INT_TO_REAL (iLiters);

END_FUNCTION_BLOCK

// POUs/PLC/Elements/MeterCounter
FUNCTION_BLOCK MeterCounter
(*************************************************************
Convert an speed input into meters - 01/12/2021
V1.00
*************************************************************)
VAR_INPUT
	xMachineRunning:BOOL;
	xFabricPresence:BOOL;
	xReset:BOOL;
	rSpeed:REAL;
END_VAR
VAR_OUTPUT
	rMeters:REAL;
END_VAR
VAR
	ContarMetros: BOOL;
	Acumulador: ContadorRapid;
	cumulado: BOOL;
	acumulado: REAL;
	acumuladoInicial: REAL;
	acumuladofinal: REAL;
	Pulsocontador: F_TRIG;
	Acumular: BOOL;
END_VAR

ContarMetros := xMachineRunning AND xFabricPresence;

Pulsocontador(CLK:=ContarMetros , Q=>Acumular);

IF Acumular
	THEN
		acumuladoInicial := acumuladofinal;
END_IF

IF xReset
	THEN
		acumuladoInicial :=0;
		acumuladofinal :=0;
END_IF

Acumulador(bActivate:=ContarMetros AND NOT xReset , rFequency:=rSpeed , rCounter_REAL=>acumulado , dwCounter_DWORD=> );

acumuladofinal := acumulado + acumuladoInicial;

rMeters := acumuladofinal/60;

END_FUNCTION_BLOCK

// POUs/PLC/Utils/Counters/ContadorRapid
FUNCTION_BLOCK ContadorRapid
(**********************************************************
Creat an totalizer from an frequency input - 26/11/2021
V1.00
*********************************************************)
VAR_INPUT
	bActivate:BOOL;			// Start executing the function
	rFequency:REAL;			// Input Frequency
END_VAR

VAR_OUTPUT
	rCounter_REAL:REAL;
	dwCounter_DWORD:DWORD;
END_VAR

VAR
	Periodecicle:Tcicle;
	ov: BOOL;
	INTEG: INTEGRAL;
END_VAR



INTEG(
	IN:=rFequency , 
	TM:=Periodecicle.dwPeriode_Cicle , 
	RESET:= ov OR NOT bActivate , 
	OUT=> rCounter_REAL, 
	OVERFLOW=> ov);

dwCounter_DWORD := REAL_TO_DWORD(rCounter_REAL);

END_FUNCTION_BLOCK

// POUs/PLC/Elements/PulseTrain
FUNCTION_BLOCK PulseTrain
(******************************************************
Generate a Pulse Train based on a % input - 10/12/2021
V1.00
*******************************************************)
VAR_INPUT
	rPorcentatge:REAL;			// Percentual Input (0-100%)
	rPeriode_seg:REAL;			// Period Input (sec)
	rPols_min_ms:REAL;			// Minimum duration of the pulse output (ms)
END_VAR

VAR_OUTPUT
	xT_Pulsos:BOOL;				// Pulse Output
END_VAR

VAR
	PararTren: BOOL;
	SegonsOFFtime: TIME;
	SegonsONtime: TIME;
	SegonsONreal: REAL;
	SegonsOFFreal: REAL;
	AperturaPulso: REAL;
	SegonsCicles: REAL;
	Tiemposinsenal: TMP;
	tempsmin: TIME;
	toff: TON;
	TON: TON;
	PulsMin : BOOL;
	TPulsMin:TP;
END_VAR

AperturaPulso := rPorcentatge;
SegonsCicles := rPeriode_seg;

SegonsONreal := (SegonsCicles*AperturaPulso)/100;
SegonsOFFreal := SegonsCicles-SegonsONreal;

SegonsONtime := REAL_TO_TIME(SegonsONreal*1000);
SegonsOFFtime := REAL_TO_TIME(SegonsOFFreal*1000);

IF SegonsONreal = 0
	THEN
		Tiemposinsenal.xIN := TRUE;
	ELSE
		Tiemposinsenal.xIN := FALSE;
END_IF

Tiemposinsenal(xIN:= , dwSegons:=5 , xQ=>PararTren , dwTsegons=> );
tempsmin := REAL_TO_TIME (rPols_min_ms);

// Generador de pulsos
toff(IN:= NOT ton.Q, PT:=SegonsOFFtime , Q=> , ET=> );
ton(IN:= toff.Q, PT:=SegonsONtime , Q=> , ET=> );

// Utiliza el pulso minimo si el tON es mas pequeno que el pulso minimo
IF SegonsONreal <= rPols_min_ms/1000
	THEN
		PulsMin := TRUE;
	ELSE
		PulsMin := FALSE;
END_IF

TPulsMin(IN:=PulsMin AND  toff.Q, PT:=tempsmin , Q=> , ET=> );

xT_Pulsos := (toff.Q AND NOT PararTren) OR (PulsMin AND TPulsMin.Q);

END_FUNCTION_BLOCK

// POUs/PLC/Elements/Washing_HT
FUNCTION_BLOCK Washing_HT
(**************************************************************
Execute a continuos washing in high temperature - 01/12/2021
V1.00
***************************************************************)
VAR_INPUT
	xStartDrain : BOOL;					// Enable the function
	xDirectDrain:BOOL;					// Enable direct drain input
	dwTimeFillAuxTank: DWORD;			// Time to transfer from machine to auxiliar tank
	dwTimeCloseAuxTank:DWORD;			// Time to finish the transfering to the auxiliar tank
	dwTimeDepAuxTank:DWORD;				// Time do depressurize auxiliar tank
	dwTimeDrainAunxTank:DWORD;			// Time to drain the auxiliar tank
	dwTimeCloseDrainAuxTank:DWORD;		// Time to garantee that the drain valve has closed
	xAlarmPauseWash:BOOL;				// Alarm Input to stop the function
	
END_VAR

VAR_OUTPUT
	xFillAuxTank:BOOL;					// Transfer from machuine to auxiliar tank
	xDepAuxTank:BOOL;					// depressurize auxiliar tank
	xDrainAuxTank:BOOL;					// Drain auxiliar tank
END_VAR

VAR
	ObrirBuidatRBB: BOOL;
	TempoPas1: TMP;
	TempoPas2: TMP;
	ObrirDespresuritzaRBB: BOOL;
	TempoPas3: TMP;
	ObrirOmplertaRBB: BOOL;
	TancarOmpertaRBB: BOOL;
	TancarBuidatRBB: BOOL;
	FiSequenciaRBB: BOOL;
	TempoPas4: TMP;
	TempoPas5: TMP;
	TemoDespesuritzaRBB: TMP;
	RBBsensePresio: BOOL;
	ObrirRespiraderoRBB: BOOL;
	FiBuidatRBB: BOOL;
	FiBuidatDirecte: F_TRIG;
	PolsFiBuidat: BOOL;
	TempSfINAL: TMP;
	ObrirBuidatAlBuidat: BOOL;
	srObrirOmplertaRBB :SR;
	srObrirRespiraderoRBB:SR;
	srPolsFiBuidat:SR;
	rtBuidatDirecte:F_TRIG;
	
	
END_VAR

// **************** Inicia el ciclo **************************
srObrirOmplertaRBB(SET1:= xStartDrain AND NOT srObrirOmplertaRBB.Q1 , RESET:=xAlarmPauseWash OR (FiSequenciaRBB AND ObrirOmplertaRBB) , Q1=>ObrirOmplertaRBB );


// **************** Temps por cada pas ************************
TempoPas1(xIN:=ObrirOmplertaRBB , dwSegons:=dwTimeFillAuxTank , xQ=>TancarOmpertaRBB , dwTsegons=> );

TempoPas2(xIN:=TancarOmpertaRBB , dwSegons:=dwTimeCloseAuxTank , xQ=>ObrirDespresuritzaRBB , dwTsegons=> );

TempoPas3(xIN:=ObrirDespresuritzaRBB , dwSegons:=dwTimeDepAuxTank , xQ=>ObrirBuidatRBB , dwTsegons=> );

TempoPas4(xIN:=ObrirBuidatRBB , dwSegons:=dwTimeDrainAunxTank , xQ=>TancarBuidatRBB , dwTsegons=> );

TempoPas5(xIN:=TancarBuidatRBB , dwSegons:=dwTimeCloseDrainAuxTank , xQ=>FiSequenciaRBB , dwTsegons=> );


srObrirRespiraderoRBB(SET1:=xDirectDrain AND NOT srObrirRespiraderoRBB.Q1, RESET:=xAlarmPauseWash OR (FiBuidatRBB AND ObrirRespiraderoRBB) , Q1=>ObrirRespiraderoRBB );

TemoDespesuritzaRBB(xIN:=ObrirRespiraderoRBB , dwSegons:=dwTimeDepAuxTank , xQ=>RBBsensePresio , dwTsegons=> );

rtBuidatDirecte(CLK:=xDirectDrain , Q=> );
srPolsFiBuidat(SET1:=rtBuidatDirecte.Q , RESET:=FiBuidatRBB , Q1=>PolsFiBuidat );

TempSfINAL(xIN:=PolsFiBuidat , dwSegons:=5 , xQ=>FiBuidatRBB , dwTsegons=> );

ObrirBuidatAlBuidat := xDirectDrain AND NOT FiBuidatRBB;

///*************************** Activa salidas ******************************
xFillAuxTank := (ObrirOmplertaRBB AND NOT TancarOmpertaRBB AND NOT xAlarmPauseWash) OR (xDirectDrain AND RBBsensePresio);

xDepAuxTank := (ObrirDespresuritzaRBB AND NOT TancarBuidatRBB AND NOT xAlarmPauseWash) OR xDirectDrain;

xDrainAuxTank := (ObrirBuidatRBB AND NOT TancarBuidatRBB AND NOT xAlarmPauseWash) OR ObrirBuidatAlBuidat;

END_FUNCTION_BLOCK

// POUs/PLC/Fill/TemperatureFill
FUNCTION_BLOCK TemperatureFill
(**********************************************************
Fill with a Temperature SetPoint - 30/11/2021
V1.00
*********************************************************)
VAR_INPUT
	xActiv			:	BOOL;		//Enable the temperature control
	rTempSP			:	REAL;		// Temperature SetPoint
	rTempPV			:	REAL;		// Real Temperature 
	rDBHigh			:	REAL;		// Superior DeadBand 
	rDBLow			:	REAL;		// Inferior DeadBand 
	timMaxTime		:	TIME;		//	Maximum time for adjust the temperature
	dwConfigMaxTime:	DWORD;		//	Maximum time configure (1 - Open just cold water, 0 - Open cold and hot water, 2 - Activate Alarm)
	xLevel			:	BOOL;		// Minimum level input
	dwConfigLevel	:	DWORD;		// Level Configure (0 - Disable, 1 - Starts filing with CW and HW, 2 - Starts filing with CW, 3 - Starts filing with HW) 
	timControl		:	TIME;		// Time delay for start adjusting the teperature.
END_VAR
VAR_OUTPUT
	xCWater				:	BOOL;	// Cold Water Output
	xHWater				:	BOOL;	// Hot Water Output
	xAlarmMaxTime		:	BOOL;	// Maximum time alarm Output
END_VAR
VAR
	TempIni 			:	TON;	
	MaxTemp 			:	TON;
	TemperMin			:	REAL;		// Temperatura mínima SP-DBmin	
	TemperMax			:	REAL;		// Temperatura mínima SP+DBmax
		
	CtrlNivel: BOOL;
END_VAR

MaxTemp(IN:=xActiv AND (rTempPV < TemperMin OR rTempPV > TemperMax) AND TempIni.Q AND SEL(CtrlNivel, 1,xLevel)  , PT:=timMaxTime , Q=>xAlarmMaxTime , ET=> );
TempIni(IN:=xActiv, PT:=timControl , Q=> , ET=> );

TemperMax := rTempSP + rDBHigh;
TemperMin := rTempSP - rDBLow;

IF dwConfigLevel > 0
	THEN
		CtrlNivel := TRUE;
	ELSE
		CtrlNivel := FALSE;
END_IF
	

IF xActiv
	THEN
		IF (rTempPV < TemperMax AND rTempPV > TemperMin AND NOT MaxTemp.Q) OR (MaxTemp.Q AND dwConfigMaxTime = 0 AND dwConfigMaxTime <> 2) OR NOT TempIni.Q OR (dwConfigLevel = 1 AND NOT xLevel) 
			THEN
				xCWater :=TRUE;
				xHWater :=TRUE;
		END_IF	
		IF rTempPV > TemperMax AND NOT MaxTemp.Q AND TempIni.Q OR (MaxTemp.Q AND dwConfigMaxTime = 1 AND dwConfigMaxTime <> 2) OR (dwConfigLevel = 3 AND NOT xLevel)
			THEN			
				xCWater :=TRUE;
				xHWater :=FALSE;			
		END_IF 
		IF rTempPV < TemperMin AND NOT MaxTemp.Q AND TempIni.Q OR (dwConfigLevel = 2 AND NOT xLevel)
			THEN			
				xCWater :=FALSE;
				xHWater :=TRUE;			
		END_IF
		IF MaxTemp.Q AND dwConfigMaxTime = 2
			THEN
				xCWater :=FALSE;
				xHWater :=FALSE;
		END_IF
	 ELSE
		xCWater :=FALSE;
		xHWater :=FALSE;			
END_IF

END_FUNCTION_BLOCK

// POUs/PLC/Utils/AnalogConversions/Canvi_Escala
FUNCTION Canvi_Escala:REAL
(**************************************************************
Execute an SCALE from an input value (REAL). If not defined
 the scales, the default values are going to be 0 (min) and 100 (max)
for both, input and output. 26/11/2021
V1.00
***************************************************************)
VAR_INPUT
	rIn:REAL;						// Input Variable
	rIn_Min:REAL:=0;				// Input Low Value
	rIn_Max:REAL:=100;				// Input High Value
	rOut_Min:REAL:=0;				// Output Low Value
	rOut_Max:REAL:=100;				// Output High Value
END_VAR

VAR
	Din: REAL;
	Dout: REAL;
END_VAR

IF rin<rin_Min
	THEN
		rin:=rin_min;
END_IF
IF rin>rin_Max
	THEN
		rin:=rin_max;
END_IF

Din:=rIn_Max-rIn_Min;

IF Din=0
	THEN
		Canvi_Escala:=0;
	ELSE
		Dout:=rOut_Max-rOut_Min;
		Canvi_Escala:=(((rIn-rIn_Min)/Din)*Dout)+rOut_Min;
END_IF

END_FUNCTION

// POUs/PLC/Utils/AnalogConversions/Conv_Temp
FUNCTION Conv_Temp:REAL
(**************************************************************** 
 Convert an temperature input (INT * 10) to an REAL value (with decimals).  26/11/2021
 V1.00
*****************************************************************)
VAR_INPUT
	wLecturaTemperatura:WORD;				//Temperature Input (WORD)
END_VAR

VAR

END_VAR

Conv_Temp:= (WORD_TO_REAL(wLecturaTemperatura))/10;

END_FUNCTION

// POUs/PLC/Utils/BitsConversions/Bits_to_Dword
FUNCTION_BLOCK Bits_to_Dword
(**********************************************************
Join 32 bits in a DWORD Variable  - 29/11/2021
V1.0
*********************************************************)
VAR_INPUT
	bBB0:BOOL;		//LSB BYTE 0
	bBB1:BOOL;
	bBB2:BOOL;
	bBB3:BOOL;
	bBB4:BOOL;
	bBB5:BOOL;
	bBB6:BOOL;
	bBB7:BOOL;		//MSB BYTE 0
	bBA0:BOOL;		//LSB BYTE 1
	bBA1:BOOL;
	bBA2:BOOL;
	bBA3:BOOL;
	bBA4:BOOL;
	bBA5:BOOL;
	bBA6:BOOL;
	bBA7:BOOL;		//MSB BYTE 1
	bAB0:BOOL;		//LSB BYTE 2
	bAB1:BOOL;		
	bAB2:BOOL;
	bAB3:BOOL;
	bAB4:BOOL;
	bAB5:BOOL;
	bAB6:BOOL;
	bAB7:BOOL;		//MSB BYTE 2
	bAA0:BOOL;		//LSB BYTE 3
	bAA1:BOOL;
	bAA2:BOOL;
	bAA3:BOOL;
	bAA4:BOOL;
	bAA5:BOOL;
	bAA6:BOOL;
	bAA7:BOOL;		//MSB BYTE 3
END_VAR

VAR_OUTPUT
	dwDW:DWORD;		// Output DWORD
END_VAR

VAR
	PART_BAIXA_BAIXA: BYTE;
	PART_BAIXA_ALTA: BYTE;
	PART_ALTA_BAIXA: BYTE;
	PART_ALTA_ALTA: BYTE;

	WORD_ALTA: WORD;
	WORD_BAIXA: WORD;
END_VAR

PART_BAIXA_BAIXA := PACK(
	B0:= bBB0, 
	B1:= bBB1, 
	B2:= bBB2, 
	B3:= bBB3, 
	B4:= bBB4, 
	B5:= bBB5, 
	B6:= bBB6, 
	B7:= bBB7);
	
PART_BAIXA_ALTA := PACK(
	B0:= bBA0,
	B1:= bBA1, 
	B2:= bBA2, 
	B3:= bBA3, 
	B4:= bBA4, 
	B5:= bBA5, 
	B6:= bBA6, 
	B7:= bBA7);
		
PART_ALTA_BAIXA := PACK(
	B0:= bAB0,
	B1:= bAB1, 
	B2:= bAB2, 
	B3:= bAB3, 
	B4:= bAB4, 
	B5:= bAB5, 
	B6:= bAB6, 
	B7:= bAB7);
	
PART_ALTA_ALTA := PACK(
	B0:= bAA0,
	B1:= bAA1, 
	B2:= bAA2, 
	B3:= bAA3, 
	B4:= bAA4, 
	B5:= bAA5, 
	B6:= bAA6, 
	B7:= bAA7);
	
WORD_BAIXA := BYTE_TO_WORD(PART_BAIXA_BAIXA) OR SHL(BYTE_TO_WORD(PART_BAIXA_ALTA),8); 
WORD_ALTA := BYTE_TO_WORD(PART_ALTA_BAIXA) OR SHL(BYTE_TO_WORD(PART_ALTA_ALTA),8); 
dwDW := WORD_TO_DWORD(WORD_BAIXA) OR SHL(WORD_TO_DWORD(WORD_ALTA),16);

END_FUNCTION_BLOCK

// POUs/PLC/Utils/BitsConversions/Bits_to_word
FUNCTION_BLOCK Bits_to_word
(**********************************************************
Join 16 bits in a WORD Variable  - 29/11/2021
V1.0
*********************************************************)

VAR_INPUT
	bB0:BOOL;		//LSB BYTE 0
	bB1:BOOL;
	bB2:BOOL;
	bB3:BOOL;
	bB4:BOOL;
	bB5:BOOL;
	bB6:BOOL;
	bB7:BOOL;		//MSB BYTE 0
	bA0:BOOL;		//LSB BYTE 1
	bA1:BOOL;
	bA2:BOOL;
	bA3:BOOL;
	bA4:BOOL;
	bA5:BOOL;
	bA6:BOOL;
	bA7:BOOL;		//MSB BYTE 1
END_VAR

VAR_OUTPUT
	wW:WORD;			//WORD Output
END_VAR

VAR
	PARTBAIXA: BYTE;
	PARTALTA: BYTE;
	WORDALTA: WORD;
END_VAR

PARTBAIXA:= PACK(
	B0:= bB0, 
	B1:= bB1, 
	B2:= bB2, 
	B3:= bB3, 
	B4:= bB4, 
	B5:= bB5, 
	B6:= bB6, 
	B7:= bB7);
	
PARTALTA:= PACK(
	B0:= bA0, 
	B1:= bA1, 
	B2:= bA2, 
	B3:= bA3, 
	B4:= bA4, 
	B5:= bA5, 
	B6:= bA6, 
	B7:= bA7);
	
WORDALTA := SHL(BYTE_TO_WORD(PARTALTA),8); 
wW := BYTE_TO_WORD(PARTBAIXA)OR WORDALTA;

END_FUNCTION_BLOCK

// POUs/PLC/Utils/BitsConversions/Dword_to_bits
FUNCTION_BLOCK Dword_to_bits
(**********************************************************
Convert a DWORD variable to 32 bits - 29/11/2021
V1.0 
*********************************************************)

VAR_INPUT
	dwDW:DWORD;		//DWORD Input
END_VAR

VAR_OUTPUT
	bBB0:BOOL;		//LSB BYTE 0
	bBB1:BOOL;
	bBB2:BOOL;
	bBB3:BOOL;
	bBB4:BOOL;
	bBB5:BOOL;
	bBB6:BOOL;
	bBB7:BOOL;		//MSB BYTE 0
	bBA0:BOOL;		//LSB BYTE 1
	bBA1:BOOL;
	bBA2:BOOL;
	bBA3:BOOL;
	bBA4:BOOL;
	bBA5:BOOL;
	bBA6:BOOL;
	bBA7:BOOL;		//MSB BYTE 1
	bAB0:BOOL;		//LSB BYTE 2
	bAB1:BOOL;
	bAB2:BOOL;
	bAB3:BOOL;
	bAB4:BOOL;
	bAB5:BOOL;
	bAB6:BOOL;
	bAB7:BOOL;		//MSB BYTE 2
	bAA0:BOOL;		//LSB BYTE 3
	bAA1:BOOL;
	bAA2:BOOL;
	bAA3:BOOL;
	bAA4:BOOL;
	bAA5:BOOL;
	bAA6:BOOL;
	bAA7:BOOL;		//MSB BYTE 3
END_VAR

VAR

END_VAR



bBB0 := EXTRACT (X:= dwDW, N:=0);
bBB1 := EXTRACT (X:= dwDW, N:=1);
bBB2 := EXTRACT (X:= dwDW, N:=2);
bBB3 := EXTRACT (X:= dwDW, N:=3);
bBB4 := EXTRACT (X:= dwDW, N:=4);
bBB5 := EXTRACT (X:= dwDW, N:=5);
bBB6 := EXTRACT (X:= dwDW, N:=6);
bBB7 := EXTRACT (X:= dwDW, N:=7);
bBA0 := EXTRACT (X:= dwDW, N:=8);
bBA1 := EXTRACT (X:= dwDW, N:=9);
bBA2 := EXTRACT (X:= dwDW, N:=10);
bBA3 := EXTRACT (X:= dwDW, N:=11);
bBA4 := EXTRACT (X:= dwDW, N:=12);
bBA5 := EXTRACT (X:= dwDW, N:=13);
bBA6 := EXTRACT (X:= dwDW, N:=14);
bBA7 := EXTRACT (X:= dwDW, N:=15);
bAB0 := EXTRACT (X:= dwDW, N:=16);
bAB1 := EXTRACT (X:= dwDW, N:=17); 
bAB2 := EXTRACT (X:= dwDW, N:=18);
bAB3 := EXTRACT (X:= dwDW, N:=19);
bAB4 := EXTRACT (X:= dwDW, N:=20);
bAB5 := EXTRACT (X:= dwDW, N:=21);
bAB6 := EXTRACT (X:= dwDW, N:=22);
bAB7 := EXTRACT (X:= dwDW, N:=23);
bAA0 := EXTRACT (X:= dwDW, N:=24);
bAA1 := EXTRACT (X:= dwDW, N:=25);
bAA2 := EXTRACT (X:= dwDW, N:=26);
bAA3 := EXTRACT (X:= dwDW, N:=27);
bAA4 := EXTRACT (X:= dwDW, N:=28);
bAA5 := EXTRACT (X:= dwDW, N:=29);
bAA6 := EXTRACT (X:= dwDW, N:=30);
bAA7 := EXTRACT (X:= dwDW, N:=31);

END_FUNCTION_BLOCK

// POUs/PLC/Utils/BitsConversions/Word_to_bits
FUNCTION_BLOCK word_to_bits
(**********************************************************
Convert a WORD variable to 16 bits - 29/11/2021
V1.0 
*********************************************************)
VAR_INPUT
	wW:WORD;			// WORD Input
END_VAR

VAR_OUTPUT
	bB0:BOOL;		//LSB BYTE 0
	bB1:BOOL;
	bB2:BOOL;
	bB3:BOOL;
	bB4:BOOL;
	bB5:BOOL;
	bB6:BOOL;
	bB7:BOOL;		//MSB BYTE 0
	bA0:BOOL;		//LSB BYTE 1
	bA1:BOOL;
	bA2:BOOL;
	bA3:BOOL;
	bA4:BOOL;
	bA5:BOOL;
	bA6:BOOL;
	bA7:BOOL;		//MSB BYTE 1
END_VAR

VAR

END_VAR

bB0 := EXTRACT (X:= wW, N:=0);
bB1 := EXTRACT (X:= wW, N:=1);
bB2 := EXTRACT (X:= wW, N:=2);
bB3 := EXTRACT (X:= wW, N:=3);
bB4 := EXTRACT (X:= wW, N:=4);
bB5 := EXTRACT (X:= wW, N:=5);
bB6 := EXTRACT (X:= wW, N:=6);
bB7 := EXTRACT (X:= wW, N:=7);
bA0 := EXTRACT (X:= wW, N:=8);
bA1 := EXTRACT (X:= wW, N:=9);
bA2 := EXTRACT (X:= wW, N:=10);
bA3 := EXTRACT (X:= wW, N:=11);
bA4 := EXTRACT (X:= wW, N:=12);
bA5 := EXTRACT (X:= wW, N:=13);
bA6 := EXTRACT (X:= wW, N:=14);
bA7 := EXTRACT (X:= wW, N:=15);

END_FUNCTION_BLOCK

// POUs/PLC/Utils/Counters/Calcul_Frequencia
FUNCTION_BLOCK Calcul_Frequencia
(**********************************************************
Calculate an counter frequency - 26/11/2021
V1.00
*********************************************************)
VAR_INPUT
	xStart:BOOL; 		// Start executing the function
	rCounter:REAL;		// Input of the counter value
END_VAR

VAR_OUTPUT
	rFrequency_REAL:REAL;		//Frequency Output (REAL)
	dwFrequency_DWORD:DWORD;		//Frequency Output (DWORD)
END_VAR

VAR
	TempoContador: TON;
	tempsConta: TIME;
	div2: REAL;
	zr: BOOL;
	cum: REAL;
	adiv: REAL;
	hz: REAL;
END_VAR

TempoContador(IN:=xStart , PT:=T#7D, Q=> , ET=>tempsConta);

div2 := TIME_TO_REAL(tempsConta);

IF	div2 = 0 
	THEN
		zr := TRUE;
	ELSE
		zr := FALSE;
END_IF

IF zr 
	THEN
		cum := RCounter;
END_IF

adiv := (RCounter - cum);

IF NOT zr 
	THEN
		hz := (1000*(adiv/div2));
	ELSE
		hz := 0;
END_IF

rFrequency_REAL := hz;
dwFrequency_DWORD := REAL_TO_DWORD(hz);

END_FUNCTION_BLOCK

// POUs/PLC/Utils/FreqCycle/CalcFreq
FUNCTION_BLOCK CalcFreq
(**********************************************************
 - 29/11/2021
V1.00
*********************************************************)

VAR_INPUT

END_VAR

VAR_OUTPUT
	wFreq:WORD;			//Frrequency Output
END_VAR

VAR
	tempor1:TON;
	pols: BOOL;
	c: WORD;
	b: WORD;
END_VAR

tempor1 (in:=NOT(tempor1.Q), PT:=t#1s, Q=>pols);

IF pols=TRUE
	THEN
	c:=a-b;
	IF a>=9999
		THEN
		a:=0;
	END_IF
	b:=a;
END_IF

wFreq:=C;

END_FUNCTION_BLOCK

// POUs/PLC/Utils/Timers/TMPpausa
FUNCTION_BLOCK TMPpausa
(**********************************************************
Timer in seconds (DWORD input) and an pause Input - 29/11/2021
V1.0
*********************************************************)
VAR_INPUT
	xIN:BOOL;				// Enable Input
	xPausa:BOOL;			// Pause Input
	dwSegons:DWORD;			// Setpoint Time in seconds (DWORD)
END_VAR
VAR_OUTPUT					
	xQ:BOOL;				// Boolean Output
	dwTsegons:DWORD;		// ET time in seconds(DWORD)
END_VAR

VAR
	TEmporitz: TON;
	Temps: TIME;
	TempsTrans: TIME;
	Pols_fin: F_TRIG;
	reset: BOOL;
	Temps_contador: TIME;
	Temps_pausa: TIME;
	contgeActual: TIME;
END_VAR

Temps := REAL_TO_TIME (DWORD_TO_REAL (dwSegons)*1000);

Pols_fin(CLK:=xPausa , Q=>reset);

IF	xPausa 
	THEN
		contgeActual := TEmporitz.ET;
END_IF

IF xPausa AND contgeActual > T#0S
	THEN
		Temps_pausa:= contgeActual;
		TempsTrans := Temps_pausa + TempsTrans; 
END_IF

TEmps_contador := Temps-TempsTrans;

TEmporitz(IN:=xIn AND NOT xPausa AND NOT reset, PT:=TEmps_contador , Q=>xQ , ET=>contgeActual );

IF NOT xIn
	THEN
	TEmps_contador := t#0s;
	TempsTrans := t#0s;
	Temps_pausa:= t#0s;
END_IF

END_FUNCTION_BLOCK
